# EPICS substitutions: modules/event/evrIoc/Db/evrPatternXL04.substitutions
#
# Pattern records
file evrPatternAll.db {
#	    Device        ,  SLC Pattern Check LNK       ,  EVR/Trigger
#	                                                    Links
  pattern { DEVICE        ,        LINK4                 ,LINK5,        LINK6              , TREF , TS1ST, TS2ND }
	  { IOC:XL04:EV01 , "IOC:XL04:EV01:FANOUTSLC PP" , ""  , "IOC:XL04:EV01:FANOUT PP" , 1E06 ,   1  ,   4   }
}
# Event records
file evrEventAll.db {
  pattern { DEVICE        }
	  { IOC:XL04:EV01 }
}
